// SIMATIC S7-200 SMART project (STEP 7-Micro/WIN SMART), CPU SR40

SYMBOL_TABLE 表格 1
起动按钮             M0.0
停止按钮             M0.1
电动机              Q0.0
当前值              VW0
预设值              VW2
END_SYMBOL_TABLE

SYMBOL_TABLE 系统符号
Always_On        SM0.0    // 始终接通
First_Scan_On    SM0.1    // 仅在第一个扫描周期时接通
END_SYMBOL_TABLE

ORGANIZATION_BLOCK MAIN:OB1
TITLE=程序注释
BEGIN
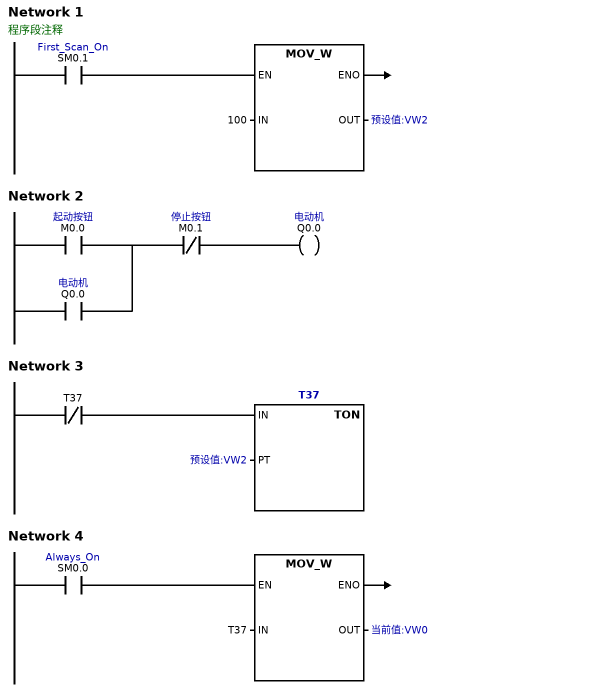
Network 1
// 程序段注释
LD     First_Scan_On:SM0.1
MOVW   100, 预设值:VW2
Network 2
LD     起动按钮:M0.0
O      电动机:Q0.0
AN     停止按钮:M0.1
=      电动机:Q0.0
Network 3
LDN    T37
TON    T37, 预设值:VW2
Network 4
LD     Always_On:SM0.0
MOVW   T37, 当前值:VW0
END_ORGANIZATION_BLOCK
